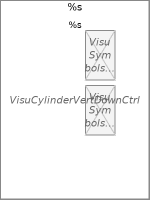
VISUALIZATION VisuCylinderVertDown  // 150x200
VAR_IN_OUT
	fbVisuCylinder: FB_VISU_CYLINDER;
END_VAR
    Image (85,85 30x50), invisible if: fbVisuCylinder.bWorkArrowInvisible, image: VisuSymbols.Symbols.ArrowBoldDown
        p2175578022: fbVisuCylinder.dwFrameColorWork
    Image (85,30 30x50), invisible if: fbVisuCylinder.bBaseArrowInvisible, image: VisuSymbols.Symbols.ArrowBoldUp
        p2175578022: fbVisuCylinder.dwFrameColorBase
    Group (25,40 40x100)
        p2738717112: fbVisuCylinder.iNegMove
        RoundedRectangle (10,0 20x100)
        RoundedRectangle (0,0 40x20)
    Rectangle (25,35 40x100)
        OnMouseClick: execute { fbVisuCylinder.bFrameInvisible:=false; }
    Textfield (0,15 150x20), "%s", text variable: fbVisuCylinder.strInfo, colour toggle: fbVisuCylinder.stEvent.bEventActive
    Textfield (0,0 150x14), "%s", text variable: fbVisuCylinder.strFullObjName
    Frame (0,0 150x200), invisible if: fbVisuCylinder.bFrameInvisible, frame switch variable: fbVisuCylinder.iFrame
        shows VisuCylinderVertDownCtrl(fbVisuCylinder := fbVisuCylinder)
END_VISUALIZATION

(* stored: Version 1.1.0.1, ProductVersion 3.1.4024.12
   Visu VisuCylinderVertDown: Id {657dd65a-e456-4064-8acb-b6f9a321095e} *)
